(* PLC project Generated.project, CODESYS CODESYS V3.5 SP19 Patch 1 *)
(* stored: creationDateTime 2026-09-14T14:47:22.329733, modificationDateTime 2026-09-14T14:47:22.329733 *)

(* ======================================================================= 🪝 ST_fbWinch_Cfg — Configuration statique d'un treuil ─────────────────────────────────────────────────────────────── 🎯 Rôle : Réglages persistants propres à l'instance treuil (statique) 📄 Doc métier : DOC/AF/AF_Partie-10_Fonction_Winch_v2.1.md 📤 Producteur : configuration persistante 📥 Consommateur : FB_Winch (statique uniquement) 🔒 Structs cibles + champs conservés pour garder le décodage %→palier et les deux cadences de rampe DANS FB_Winch (comportement bit-identique). Le champ StepRampDelay est déclaré mais non consommé (usage aval). ======================================================================= *)
TYPE ST_fbWinch_Cfg : STRUCT
  SpeedStepTable : ST_SpeedStepTable;  (* === TABLE DES PALIERS === Table de seuils des paliers de vitesse *)
  DirectionInterlockDelayAscent : TIME := TIME#800ms;  (* === INTERLOCK CHANGEMENT DE SENS === Delai interlock inversion vers montee *)
  DirectionInterlockDelayDescent : TIME := TIME#500ms;  (* Delai interlock inversion vers descente *)
  StepRampDelay : TIME := TIME#700ms;  (* === CADENCE DE RAMPE PALIER === [cible] Tempo de rampe palier (usage aval) *)
  StepRampDelayAscent : TIME := TIME#700ms;  (* [08a] Cadence palier montee (D10, dedie) *)
  StepRampDelayDescent : TIME := TIME#500ms;  (* [08a] Cadence palier descending (D10, dedie) *)
  ContactorFeedbackTimeout : TIME := TIME#500ms;  (* === RETOMBÉE CONTACTEURS === Delai d'attente retombee des contacteurs *)
  SlowdownDistanceTop_M : REAL := 0.5;  (* === RALENTISSEMENT BORDURE === Distance avant limite haute pour ralentir (m) : 0 = arrêt au seuil *)
  SlowdownDistanceBottom_M : REAL := 1;  (* Distance avant limite basse pour ralentir (m) *)
  SlowdownMaxStep : INT := 1;  (* Plafond palier dans zone de ralentissement (1..5) *)
  SpeedStepHystMargin : REAL := 2;  (* === DÉCODAGE %→PALIER (conservé) === [08a] Marge d'hysteresis palier (%) *)
END_STRUCT;
END_TYPE

(* ======================================================================= 🪜 ST_SpeedStepTable — Table des paliers de vitesse contacteurs ─────────────────────────────────────────────────────────────── 🎯 Rôle : Structure de configuration des contacteurs et seuils par palier 📄 Doc métier : DOC/AF/AF_Partie-10_Fonction_Winch_v2.1.md ======================================================================= *)
TYPE ST_SpeedStepTable : STRUCT
  P1R1 : BOOL;  (* === PALIER 1 (VITESSE MINIMALE) === Contacteur 1 pour Palier 1 *)
  P1R2 : BOOL;  (* Contacteur 2 pour Palier 1 *)
  P1R3 : BOOL;  (* Contacteur 3 pour Palier 1 *)
  P1R4 : BOOL;  (* Contacteur 4 pour Palier 1 *)
  P2R1 : BOOL;  (* === PALIER 2 === Contacteur 1 pour Palier 2 *)
  P2R2 : BOOL;  (* Contacteur 2 pour Palier 2 *)
  P2R3 : BOOL;  (* Contacteur 3 pour Palier 2 *)
  P2R4 : BOOL;  (* Contacteur 4 pour Palier 2 *)
  P3R1 : BOOL;  (* === PALIER 3 === Contacteur 1 pour Palier 3 *)
  P3R2 : BOOL;  (* Contacteur 2 pour Palier 3 *)
  P3R3 : BOOL;  (* Contacteur 3 pour Palier 3 *)
  P3R4 : BOOL;  (* Contacteur 4 pour Palier 3 *)
  P4R1 : BOOL;  (* === PALIER 4 === Contacteur 1 pour Palier 4 *)
  P4R2 : BOOL;  (* Contacteur 2 pour Palier 4 *)
  P4R3 : BOOL;  (* Contacteur 3 pour Palier 4 *)
  P4R4 : BOOL;  (* Contacteur 4 pour Palier 4 *)
  P5R1 : BOOL;  (* === PALIER 5 (VITESSE MAXIMALE) === Contacteur 1 pour Palier 5 *)
  P5R2 : BOOL;  (* Contacteur 2 pour Palier 5 *)
  P5R3 : BOOL;  (* Contacteur 3 pour Palier 5 *)
  P5R4 : BOOL;  (* Contacteur 4 pour Palier 5 *)
  StepThreshold_Pct : ARRAY[1..5] OF REAL;  (* === SEUILS DE TRANSITION (%) === Seuils de changement de palier (0..100%) *)
END_STRUCT;
END_TYPE
